// TIA Portal V20 export
DATA_BLOCK "RealDbName"   // DB7
   VAR RETAIN
      Inputs : Struct
         InHand : Bool;
         RunTime { S7_SetPoint := 'True'} : Real := 0.0;
         Nested : Struct
            DeepFlag : Bool;
         END_STRUCT;
      END_STRUCT;
   END_VAR
BEGIN
END_DATA_BLOCK
